{attribute 'reflection'} 
FUNCTION_BLOCK Zustandsautomat
VAR CONSTANT
	MaxProducts	: UINT := 5;
END_VAR
VAR_INPUT
	Panel				: REFERENCE TO ST_Panel;
	AddVisu				: InterfaceVisu;
	ZustandsautomatName	: STRING(255);

END_VAR
VAR
  State            		: E_States;
  Products         		: UINT := MaxProducts;
  trigButton         	: R_TRIG;
  trigInsertCoin     	: R_TRIG;
  trigTakeProduct    	: R_TRIG;
  trigTakeCoin       	: R_TRIG;


	NeuInit						: BOOL;
//only for VISU
	{attribute 'instance-path'} 
	{attribute 'no_init'} 
	InstanzZustandsautomat		: STRING(255);
 	InstanzNameZustandsautomat	: STRING(255);
END_VAR

Init();
stateMachine();
conditions();

METHOD conditions : BOOL
VAR_INPUT
END_VAR
Panel.NumberOfProducts := Products;
Panel.State := TO_STRING(State);
END_METHOD

METHOD Init : BOOL
VAR_INPUT
END_VAR
VAR
	tempName	: STRING(255);
	nDotFound	: INT;
END_VAR

IF NOT NeuInit THEN
	NeuInit:=TRUE;

	tempName:=InstanzZustandsautomat;
	nDotFound:=FIND(tempName,'.');
	WHILE nDotFound <> 0 DO
		tempName := RIGHT(tempName, LEN(tempName)-nDotFound);
		nDotFound := Tc2_Standard.FIND(tempName, '.');
	END_WHILE

	InstanzNameZustandsautomat := tempName;
	Panel.InstanzName:=InstanzNameZustandsautomat;
	
	IF ADR(Panel) <> 0 THEN
		AddVisu.ZustandsautomatAddVisu(	P_Panel:=ADR(Panel),
										Name := ZustandsautomatName);
	END_IF
								
	
END_IF
END_METHOD

METHOD stateMachine : BOOL
VAR_INPUT
END_VAR
trigButton(CLK := Panel.Button);
trigInsertCoin(CLK := Panel.InsertCoin);
trigTakeProduct(CLK := Panel.TakeProduct);
trigTakeCoin(CLK := Panel.TakeCoin);
 
CASE State OF
  E_States.Waiting:
    IF (trigButton.Q) THEN
      ; // keep in the state
    END_IF
    IF (trigInsertCoin.Q) THEN
      ADSLOGSTR(ADSLOG_MSGTYPE_HINT, 'Customer has insert a coin.', '');
      State := E_States.HasCoin;
    END_IF
 
  E_States.HasCoin:
    IF (trigButton.Q) THEN
      IF (Products > 0) THEN
        Products := Products - 1;
        ADSLOGSTR(ADSLOG_MSGTYPE_HINT, 'Customer has pressed the button. Output product.', '');
        State := E_States.ProductEjected;
      ELSE
        ADSLOGSTR(ADSLOG_MSGTYPE_HINT, 'Customer has pressed the button. No more products. Return coin.', '');
        State := E_States.CoinEjected;
      END_IF
    END_IF
 
  E_States.ProductEjected:
    IF (trigTakeProduct.Q) THEN
      ADSLOGSTR(ADSLOG_MSGTYPE_HINT, 'Customer has taken the product.', '');
      State := E_States.Waiting;
    END_IF
 
  E_States.CoinEjected:
    IF (trigTakeCoin.Q) THEN
      ADSLOGSTR(ADSLOG_MSGTYPE_HINT, 'Customer has taken the coin.', '');
      State := E_States.Waiting;
    END_IF
 
  ELSE
    ADSLOGSTR(ADSLOG_MSGTYPE_ERROR, 'Invalid state', '');
    State := E_States.Waiting;
END_CASE
END_METHOD

END_FUNCTION_BLOCK

(* stored: Version 1.1.0.1, ProductVersion 3.1.4024.9
   POU Zustandsautomat: Id {06aab81e-e47c-4303-86d6-ad89b6118069}, SpecialFunc None
   Method conditions: Id {737e76b9-6c29-4c2e-9f69-c3f0986c32ce}
   Method Init: Id {e23b1f8a-7b01-4887-ad95-8a9f68570603}
   Method stateMachine: Id {60b1a753-bb52-4aa5-b91b-89874d07573b} *)
